(* PLC project Untitled1, Beckhoff Automation GmbH TwinCAT PLC Control 3.5.13.21 *)
(* stored: creationDateTime 2025-01-07T13:20:58.3085275, modificationDateTime 2025-01-07T13:20:58.3085275 *)

FUNCTION F_TrueBitsCounter : UINT
VAR_INPUT
	pArray			: POINTER TO ARRAY[0..255] OF BOOL;
	arrBitSize		: UINT; 
END_VAR
	
VAR
	i				: UINT;
END_VAR

            

FOR i:=0 TO arrBitSize-1 DO
	IF pArray^[i] THEN
		F_TrueBitsCounter	:= F_TrueBitsCounter + 1;
	END_IF
END_FOR
          
END_FUNCTION
